{attribute 'GeneratedUsingTerminal: EL4032-0000-0018'}
{attribute addProperty BoxType "EL4032-0000-0018"}
{attribute addProperty Id "AO_Output_Channel_1AT %Q*AO_Output_Channel_BA7EBB7C2AO_Output_Channel_2AT %Q*AO_Output_Channel_BA7EBB7C2WcStateAT %I*WcState_0B2B16F91InfoDataAT %I*InfoData_32EB74EA10"}
{attribute addProperty CRC "1524858257"}
{attribute addProperty Size "15"}
TYPE EL4032_5AE37D91 EXTENDS EtcSlaveTerminalBase_947E5A46 :
STRUCT
	{attribute addProperty Name "AO_Output_Channel_1"}
	AO_Output_Channel_1 : AO_Output_Channel_BA7EBB7C;
	{attribute addProperty Name "AO_Output_Channel_2"}
	AO_Output_Channel_2 : AO_Output_Channel_BA7EBB7C;
	{attribute addProperty Name "WcState"}
	WcState : WcState_0B2B16F9;
	{attribute addProperty Name "InfoData"}
	InfoData : InfoData_32EB74EA;
END_STRUCT
END_TYPE

(* stored: Version 1.2.0.0, ProductVersion 3.1.4024.9
   DUT EL4032_5AE37D91: Id {cf831e13-2941-4067-aeec-c9e574923e1d} *)
